FUNCTION CheckDivZero : REAL
VAR_INPUT
	rInput:REAL;	(*Entrada a ser comparada*)
END_VAR
VAR
END_VAR
(*Apenas verifica se a entrada e igual a zero para poder realizar um divisao*)
(*just check if the input is zero to make a division operation*)

(*Apenas verifica se a entrada dessa funcao é igual a zero*)
IF rInput <> 0 THEN
	CheckDivZero := rInput;
ELSE
	CheckDivZero:=1;
END_IF

END_FUNCTION

(* stored: Version 1.1.0.1, ProductVersion 3.1.4024.12
   POU CheckDivZero: Id {a9f903f9-f88a-4009-a599-edd6afc82439}, SpecialFunc None *)
